INTERFACE ITF_Control

METHOD GetSwitchS10 : BOOL
VAR_INPUT
END_VAR
END_METHOD

END_INTERFACE

(* stored: Version 1.1.0.1, ProductVersion 3.1.4024.12
   Itf ITF_Control: Id {fc73c7a9-2723-46ae-8509-a5372f653e2d}
   Method GetSwitchS10: Id {03a33c3c-e9f7-4db0-a255-92f5eb3f6b3a} *)
